// SIMATIC S7-200 project (STEP 7-Micro/WIN), CPU 226 REL 02.01

SYMBOL_TABLE USR1
出水温度VF           I0.0
回水温度VF           I0.1
燃烧信号             I0.2
尾烟温度VF           I0.3
超温报警             I0.4
超高压力             I0.5
低限压力             I0.6
循环泵信号            I0.7
风机反馈             I1.0
低水位              I1.1
停炉消音             I1.2
熄火               I1.3
启动复位             I1.4
循环水泵             Q0.0
蜂鸣器              Q0.1
风机               Q0.2
减低负荷             Q0.4
加大负荷             Q0.5
锅炉运行控制           Q0.7
故障               Q1.0
第一段温度            M0.0
第二段温度            M0.1
第三段温度            M0.2
第四段温度            M0.3
第五段温度            M0.4
显示手动键            M1.4
后扫显示             M1.5
强制小火显示           M1.6
复位显示             M1.7
点火成功             M2.0
可以燃烧             M2.1
喷油标志             M2.4
进入消音             M2.6
停火消音             M2.7
手动负荷             M4.0
手动关小             M4.1
手动开大             M4.2
分段控制             M4.5
工作时间             M4.6
等待工作             M5.0
启动标志             M5.1
锅炉启动             M5.2
停火标志             M5.7
负荷减小             M6.0
负荷加大             M6.1
负荷在减小            M6.2
负荷在加大            M6.3
消音标志             M7.3
屏启动按钮            M8.0
屏停炉按钮            M8.1
屏消音按钮            M8.2
屏复位按钮            M8.3
消音脉冲             M8.5
启动脉冲             M8.6
复位脉冲             M8.7
PLC是运行           M9.0
记录清零             M9.3
停火故障             M9.6
严重故障             M9.7
报极低水位            M10.7
锅炉压力失常           M10.6
传感器故障            M10.5
报限位故障            M10.4
报超高温度            M10.3
风门关故障            M10.2
风门中继坏            M10.1
燃气压力低            M10.0
超高烟温             M11.7
点火失败             M11.6
风压不足故障           M11.5
关阀故障             M11.4
故障熄火             M11.3
故障见火             M11.2
风门开故障            M11.1
风门小故障            M11.0
要求大火             M12.2
记录小火             M12.3
动画小火             M12.4
记录大火             M12.5
动画大火             M12.6
温度启停炉            M13.1
出口传感器故障          M13.2
烟温高              M13.3
大小火控制            M13.5
设置时间             M14.0
不检传感             M14.4
管理密码对            M15.1
MODBUS1          M18.0
MODBUS2          M18.1
屏动画风机            M20.0
屏动画水泵            M20.1
强制小火             M31.1
手动开风机            M31.2
水泵自动             M31.3
水泵手动             M31.4
水泵停              M31.5
PLC运行            SM0.0
运行脉冲             SM0.1
分振荡器             SM0.4
PLC在运行           SM0.7
中断1              SMB34
中断2              SMB35
HC0控制字           SMB37
HC0当前值           SMD38
HC3控制字           SMB137
HC3当前值           SMD138
HC4控制字           SMB147
HC4当前值           SMD148
不见光极限            T34
确认点火             T37
确认停火             T38
确认小火             T42
报警延时             T49
是极低水位            T51
是超高温度            T52
是锅炉超压            T53
是欠压              T54
是传感器故障           T55
是烟温高             T56
减负荷              T101
加负荷              T102
开机3秒             T103
后吹扫控制            T112
程控小火完成           T117
报荡显示1            T130
振荡显示2            T131
开机2秒             T142
记录工时分            C15
水泵工时分            C16
风机工时分            C17
燃烧工时分            C18
时间（年）16          VB10
时间（月）16          VB11
时间（日）16          VB12
时间（时）16          VB13
时间（分）16          VB14
时间（秒）16          VB15
实际状态编码           VW18
密码确认1            VW20
密码确认2            VW22
密码确认3            VW24
密码确认4            VW26
时间分段数            VW38
后吹扫时间            VW40
强制小火时间           VW46
给定出口温度           VD50
给定出口温度W          VW52
给定尾烟温            VW54
禁改测试页号           VW58
开机密码             VW62
管理密码             VW64
输管理密码            VW66
输开机密码            VW68
MODBUS11         VB70
MODBUS21         VB71
实际工作段            VB72
屏火焰指针            VW82
故障编码             VW86
高8               VB88
低8               VB89
故障码反             VW88
出口截距             VW90
回水截距             VW92
尾烟截距             VW94
启炉温              VW96
停火温              VW98
出口斜率             VD100
回水斜率             VD104
尾烟斜率             VD108
设定停火温            VW120
设定启动温            VW122
点火次数             VW140
工时               VW142
停炉故障次            VW144
低水位故障次           VW146
熄火次数             VW148
高温停炉次            VW150
水泵工时             VW160
风机工时             VW162
燃烧工时             VW164
定时控制             VW200
积分加强             VD202
微分加强             VD212
EI               VD222
EI1              VD232
EI2              VD242
AEI              VD252
AEI1             VD262
AAEI             VD272
查EI              VD282
比例加强             VD292
负荷调节总量           VD302
比例计算             VD312
P                VD322
积分计算             VD332
I                VD342
微分计算             VD352
D                VD362
PID计算            VD372
PID              VD382
PID累加            VD392
可控PID            VD402
余下PID            VD412
正PID控制时间         VD422
加PID             VW424
剩余PID            VD432
负PID控制时间         VD442
减PID             VW444
普通出口设定温          VD900
第一时间段设定温度1       VD904
第二时间段设定温度2       VD908
第三时间段设定温度3       VD912
第四时间段设定温度4       VD916
第五时间段设定温度5       VD920
采样记数器            VW1000
实际出口温            VD1020
实际出口温W           VW1022
出口温采样值           VD1024
出口采样             VW1026
出水计算1            VD1032
出水计算1高8位         VW1032
出水计算1低8位         VW1034
出水计算2            VD1036
实际回水温            VD1040
实际回水温W           VW1042
回水温采样值           VD1044
回水采样             VW1046
回水计算1            VD1052
回水计算1高8位         VW1052
回水计算1低8位         VW1054
回水计算2            VD1056
实际尾烟温            VD1060
实际尾烟温W           VW1062
尾烟温采样值           VD1064
尾烟采样             VW1066
尾烟计算1            VD1072
尾烟计算1高8位         VW1072
尾烟计算1低8位         VW1074
尾烟计算2            VD1076
时间1开时            VW2370
时间1开分            VW2376
时间1关时            VW2390
时间1关分            VW2396
时间2开时            VW2410
时间2开分            VW2416
时间2关时            VW2430
时间2关分            VW2436
时间3开时            VW2450
时间3开分            VW2456
时间3关时            VW2470
时间3关分            VW2476
时间4开时            VW2490
时间4开分            VW2496
时间4关时            VW2510
时间4关分            VW2516
时间5开时            VW2530
时间5开分            VW2536
时间5关时            VW2550
时间5关分            VW2556
实际时间             VW2600
实际时              VW2602
实际分              VW2604
实际时转分            VW2606
开1时间             VW2610
开1时转分            VW2612
关1时间             VW2616
关1时转分            VW2618
开2时间             VW2620
开2时转分            VW2622
关2时间             VW2626
关2时转分            VW2628
开3时间             VW2630
开3时转分            VW2632
关3时间             VW2636
关3时转分            VW2638
开4时间             VW2640
开4时转分            VW2642
关4时间             VW2646
关4时转分            VW2648
开5时间             VW2650
开5时转分            VW2652
关5时间             VW2656
关5时转分            VW2658
传送首址             VB3000
传工作状态            VW3000
传极低水位            VW3002
传锅炉压力失常          VW3004
传出口传感故障          VW3006
传燃烧器限位故障         VW3008
传超高温度            VW3010
传风门关闭故障          VW3012
传风门中继故障          VW3014
传燃气压力低           VW3016
传超高烟温            VW3018
传风压不足            VW3020
传关阀故障            VW3022
传熄火故障            VW3024
传故障见火            VW3026
传风门开故障           VW3028
传风门小故障           VW3030
传后扫时间            VW3032
传强制小火时间          VW3034
传点火次数            VW3036
传工时              VW3038
传故障停炉次数          VW3040
传给定温度            VW3042
传给定烟温            VW3044
传实际烟温            VW3046
传实际出口温           VW3048
传实际回水温           VW3050
END_SYMBOL_TABLE

SYMBOL_TABLE USS Protocol
USS_LOW_V        VD1000   // (DWORD) Enter the starting address for USS Protocol symbols here.
USS_HIGH_V       VD1004
USS_TIME_OUT     VW1008
USS_I_LINE       VW1010
USS_DAT_PTR0     VD1012
USS_ACT_DRV0     VD1016
USS_CUR_DRV0     VD1020
USS_P0           V1024.0
USS_REQ_SNT0     V1024.1
USS_RETRY_P0     VB1025
USS_ERR_CODE     VB1026
USS_CS_D0        VD1027
USS_CS_W0        VW1027
USS_CS_W2        VW1029
USS_CS_B0        VB1027
USS_CS_B1        VB1028
USS_POLL_BUF     VB1031
USS_XMT_0        VB1046
USS_XMT_ADR0     VB1049
USS_X_STWD       VD1056
USS_X_BCC        VB1060
USS_X_DW1        VD1047
USS_X_DW5        VD1051
USS_X_DW9        VD1055
USS_X_DB13       VB1059
USS_RCV_BUF0     VB1061
USS_R_STX        VB1062
USS_R_LGE        VB1063
USS_R_ADR        VB1064
USS_R_STWD       VD1071
USS_R_DW1        VD1062
USS_R_DW5        VD1066
USS_R_DW9        VD1070
USS_R_W13        VW1074
USS_STAT_TAB     VB1076
USS_ADR_P0       VB1396
END_SYMBOL_TABLE

ORGANIZATION_BLOCK MAIN:OB1
TITLE= 
// PROGRAM COMMENTS
// Press F1 for help and example program
//  
BEGIN
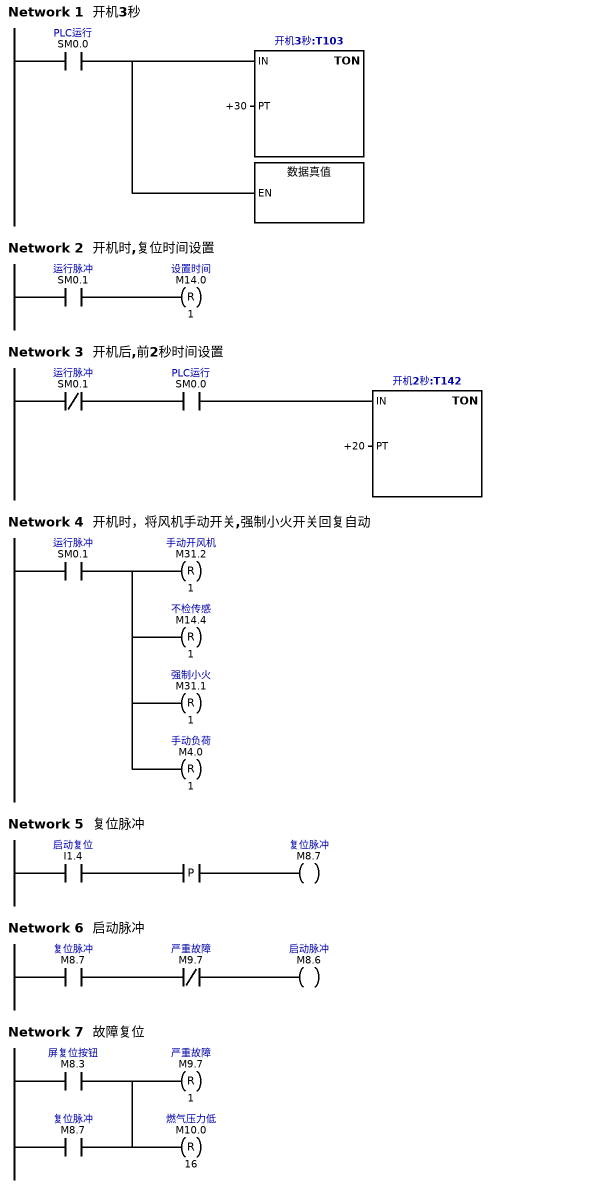
Network 1 // 开机3秒
// 
// 
LD     PLC运行:SM0.0
TON    开机3秒:T103, +30
CALL   数据真值:SBR0
Network 2 // 开机时,复位时间设置
LD     运行脉冲:SM0.1
R      设置时间:M14.0, 1
Network 3 // 开机后,前2秒时间设置
// 
// 
LDN    运行脉冲:SM0.1
A      PLC运行:SM0.0
TON    开机2秒:T142, +20
Network 4 // 开机时，将风机手动开关,强制小火开关回复自动
// 
// 
LD     运行脉冲:SM0.1
R      手动开风机:M31.2, 1
R      不检传感:M14.4, 1
R      强制小火:M31.1, 1
R      手动负荷:M4.0, 1
Network 5 // 复位脉冲
LD     启动复位:I1.4
EU
=      复位脉冲:M8.7
Network 6 // 启动脉冲
LD     复位脉冲:M8.7
AN     严重故障:M9.7
=      启动脉冲:M8.6
Network 7 // 故障复位
// 
// 
LD     屏复位按钮:M8.3
O      复位脉冲:M8.7
R      严重故障:M9.7, 1
R      燃气压力低:M10.0, 16
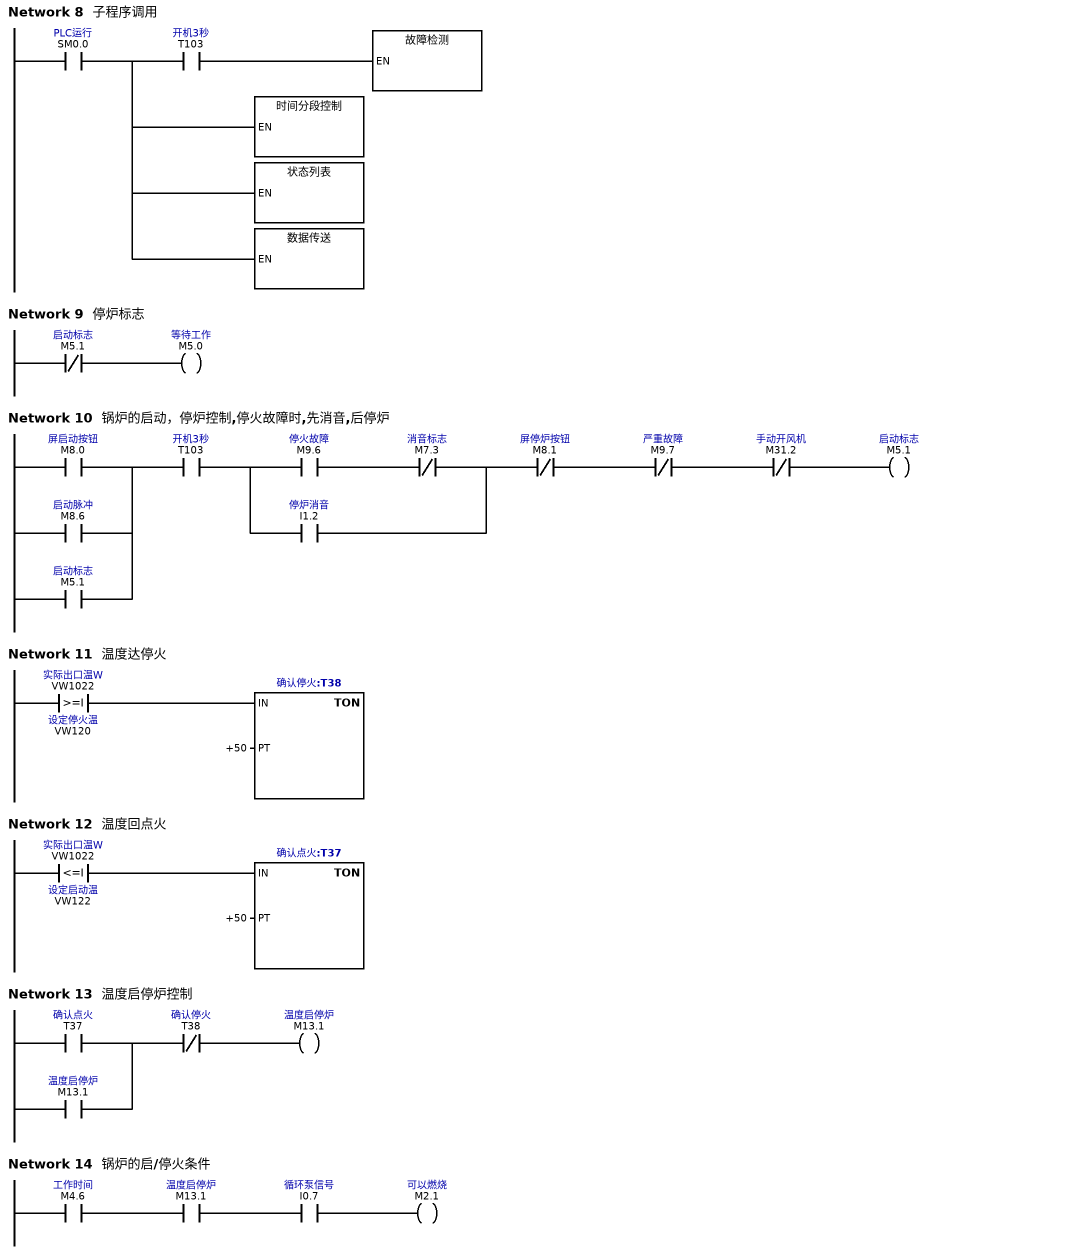
Network 8 // 子程序调用
// 
//  
LD     PLC运行:SM0.0
LPS
A      开机3秒:T103
CALL   故障检测:SBR4
LRD
CALL   时间分段控制:SBR6
LRD
CALL   状态列表:SBR7
LPP
CALL   数据传送:SBR8
Network 9 // 停炉标志
// 
// 
LDN    启动标志:M5.1
=      等待工作:M5.0
Network 10 // 锅炉的启动，停炉控制,停火故障时,先消音,后停炉
// 
// 
LD     屏启动按钮:M8.0
O      启动脉冲:M8.6
O      启动标志:M5.1
A      开机3秒:T103
LD     停火故障:M9.6
AN     消音标志:M7.3
O      停炉消音:I1.2
ALD
AN     屏停炉按钮:M8.1
AN     严重故障:M9.7
AN     手动开风机:M31.2
=      启动标志:M5.1
Network 11 // 温度达停火
// 
// 
LDW>=  实际出口温W:VW1022, 设定停火温:VW120
TON    确认停火:T38, +50
Network 12 // 温度回点火
// 
// 
LDW<=  实际出口温W:VW1022, 设定启动温:VW122
TON    确认点火:T37, +50
Network 13 // 温度启停炉控制
// 
// 
LD     确认点火:T37
O      温度启停炉:M13.1
AN     确认停火:T38
=      温度启停炉:M13.1
Network 14 // 锅炉的启/停火条件
// 
// 
LD     工作时间:M4.6
A      温度启停炉:M13.1
A      循环泵信号:I0.7
=      可以燃烧:M2.1
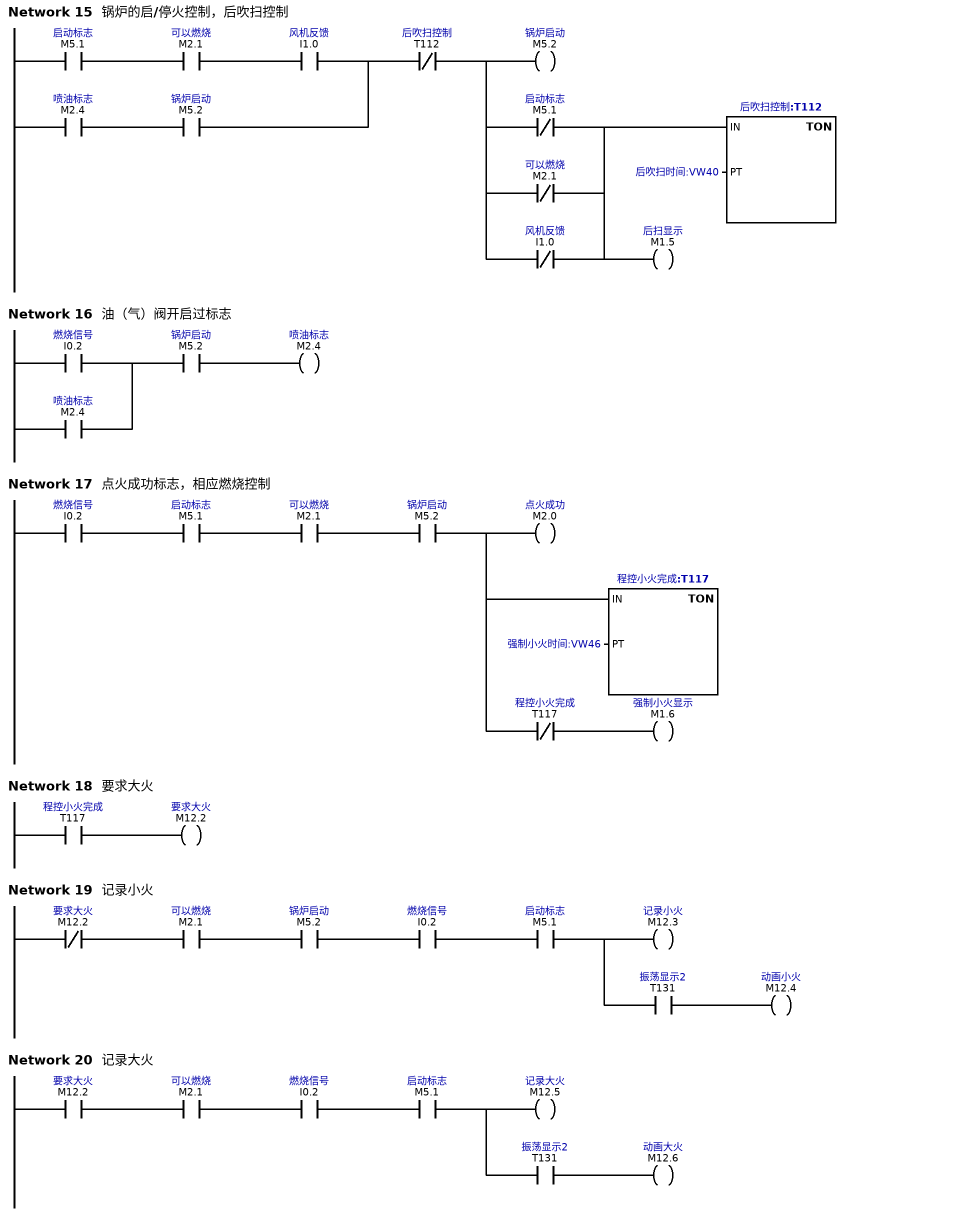
Network 15 // 锅炉的启/停火控制，后吹扫控制
// 
// 
LD     启动标志:M5.1
A      可以燃烧:M2.1
A      风机反馈:I1.0
LD     喷油标志:M2.4
A      锅炉启动:M5.2
OLD
AN     后吹扫控制:T112
=      锅炉启动:M5.2
LDN    启动标志:M5.1
ON     可以燃烧:M2.1
ON     风机反馈:I1.0
ALD
TON    后吹扫控制:T112, 后吹扫时间:VW40
=      后扫显示:M1.5
Network 16 // 油（气）阀开启过标志
// 
// 
LD     燃烧信号:I0.2
O      喷油标志:M2.4
A      锅炉启动:M5.2
=      喷油标志:M2.4
Network 17 // 点火成功标志，相应燃烧控制
// 
// 
LD     燃烧信号:I0.2
A      启动标志:M5.1
A      可以燃烧:M2.1
A      锅炉启动:M5.2
=      点火成功:M2.0
TON    程控小火完成:T117, 强制小火时间:VW46
AN     程控小火完成:T117
=      强制小火显示:M1.6
Network 18 // 要求大火
LD     程控小火完成:T117
=      要求大火:M12.2
Network 19 // 记录小火
LDN    要求大火:M12.2
A      可以燃烧:M2.1
A      锅炉启动:M5.2
A      燃烧信号:I0.2
A      启动标志:M5.1
=      记录小火:M12.3
A      振荡显示2:T131
=      动画小火:M12.4
Network 20 // 记录大火
LD     要求大火:M12.2
A      可以燃烧:M2.1
A      燃烧信号:I0.2
A      启动标志:M5.1
=      记录大火:M12.5
A      振荡显示2:T131
=      动画大火:M12.6
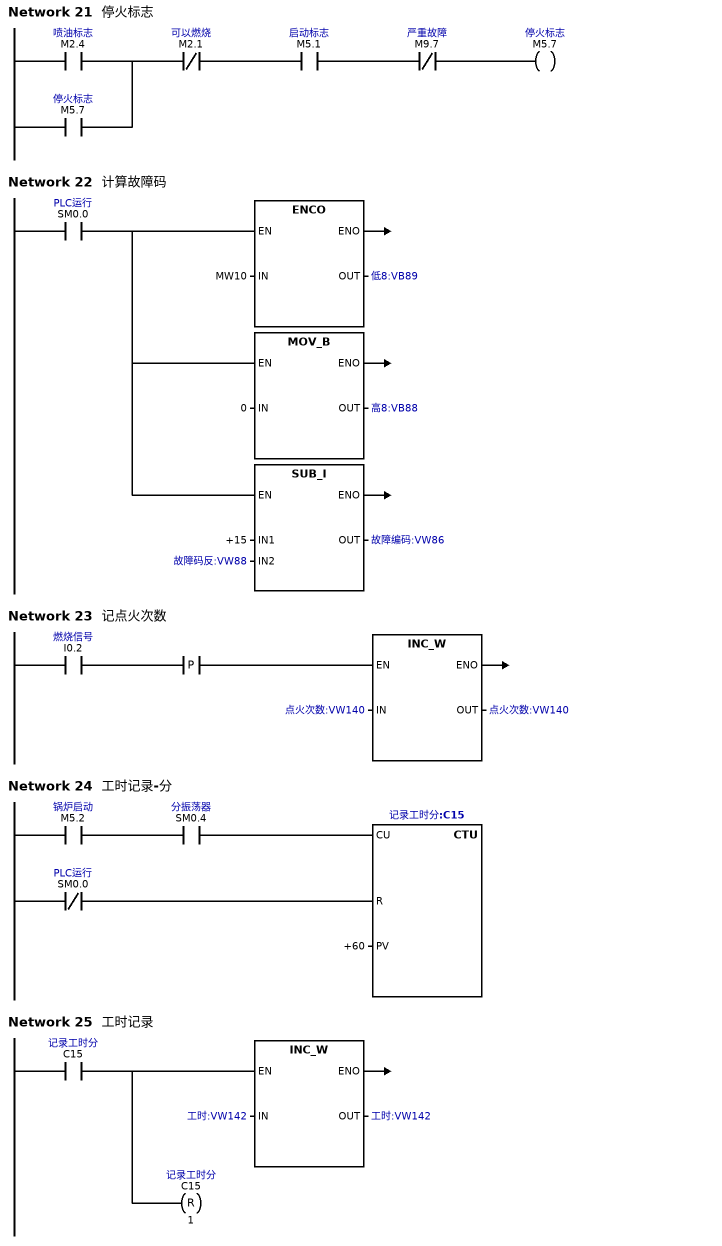
Network 21 // 停火标志
// 
// 
LD     喷油标志:M2.4
O      停火标志:M5.7
AN     可以燃烧:M2.1
A      启动标志:M5.1
AN     严重故障:M9.7
=      停火标志:M5.7
Network 22 // 计算故障码
// 
// 
LD     PLC运行:SM0.0
ENCO   MW10, 低8:VB89
MOVB   0, 高8:VB88
MOVW   +15, 故障编码:VW86
-I     故障码反:VW88, 故障编码:VW86
Network 23 // 记点火次数
// 
// 
LD     燃烧信号:I0.2
EU
INCW   点火次数:VW140
Network 24 // 工时记录-分
// 
// 
LD     锅炉启动:M5.2
A      分振荡器:SM0.4
LDN    PLC运行:SM0.0
CTU    记录工时分:C15, +60
Network 25 // 工时记录
// 
// 
LD     记录工时分:C15
INCW   工时:VW142
R      记录工时分:C15, 1
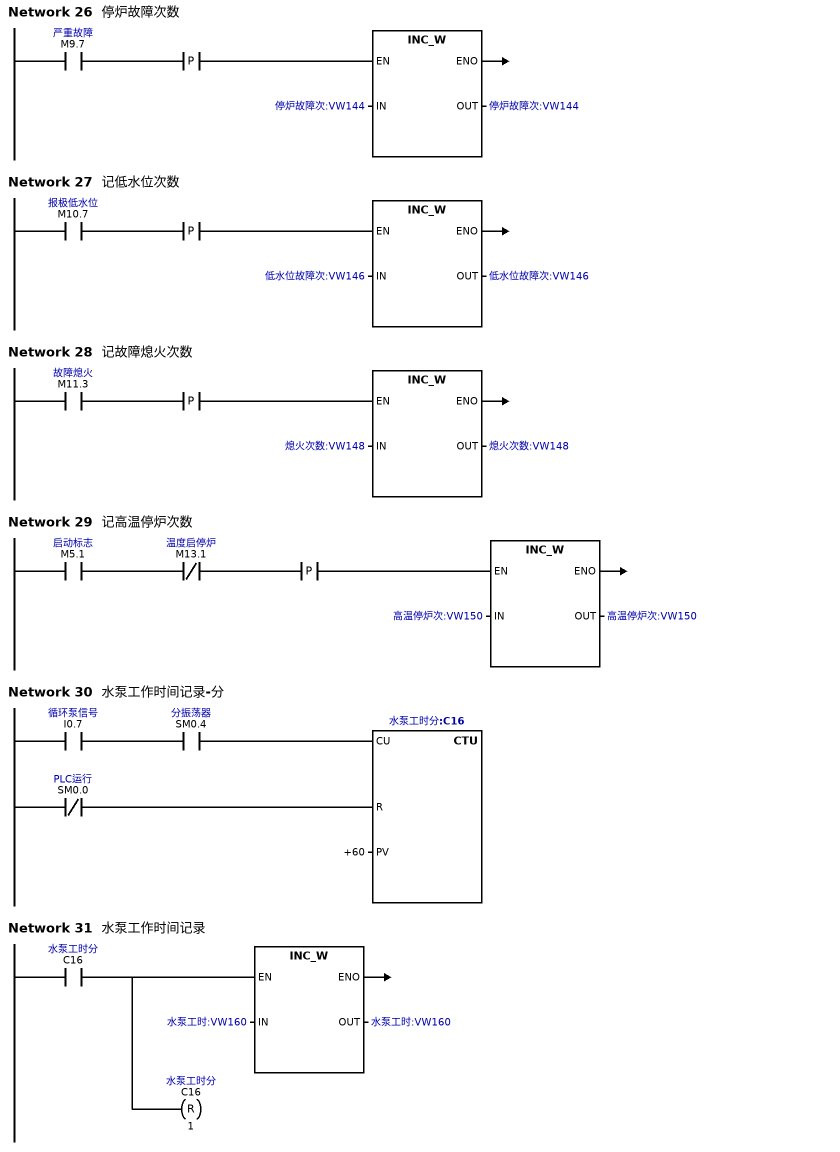
Network 26 // 停炉故障次数
// 
// 
LD     严重故障:M9.7
EU
INCW   停炉故障次:VW144
Network 27 // 记低水位次数
// 
// 
LD     报极低水位:M10.7
EU
INCW   低水位故障次:VW146
Network 28 // 记故障熄火次数
// 
// 
LD     故障熄火:M11.3
EU
INCW   熄火次数:VW148
Network 29 // 记高温停炉次数
// 
// 
LD     启动标志:M5.1
AN     温度启停炉:M13.1
EU
INCW   高温停炉次:VW150
Network 30 // 水泵工作时间记录-分
// 
// 
LD     循环泵信号:I0.7
A      分振荡器:SM0.4
LDN    PLC运行:SM0.0
CTU    水泵工时分:C16, +60
Network 31 // 水泵工作时间记录
// 
// 
LD     水泵工时分:C16
INCW   水泵工时:VW160
R      水泵工时分:C16, 1
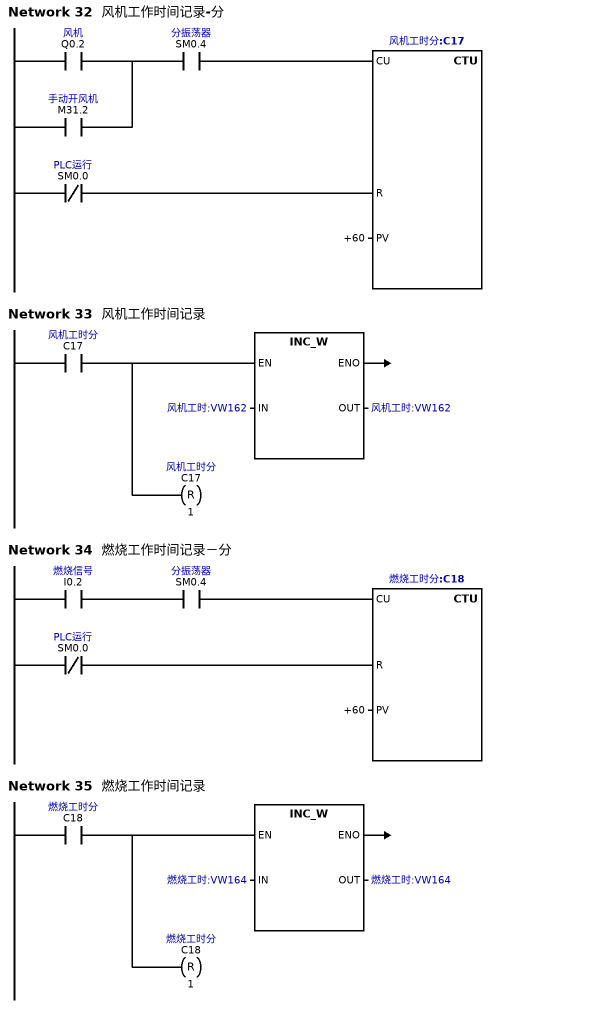
Network 32 // 风机工作时间记录-分
// 
// 
LD     风机:Q0.2
O      手动开风机:M31.2
A      分振荡器:SM0.4
LDN    PLC运行:SM0.0
CTU    风机工时分:C17, +60
Network 33 // 风机工作时间记录
// 
// 
LD     风机工时分:C17
INCW   风机工时:VW162
R      风机工时分:C17, 1
Network 34 // 燃烧工作时间记录－分
// 
// 
LD     燃烧信号:I0.2
A      分振荡器:SM0.4
LDN    PLC运行:SM0.0
CTU    燃烧工时分:C18, +60
Network 35 // 燃烧工作时间记录
// 
// 
LD     燃烧工时分:C18
INCW   燃烧工时:VW164
R      燃烧工时分:C18, 1
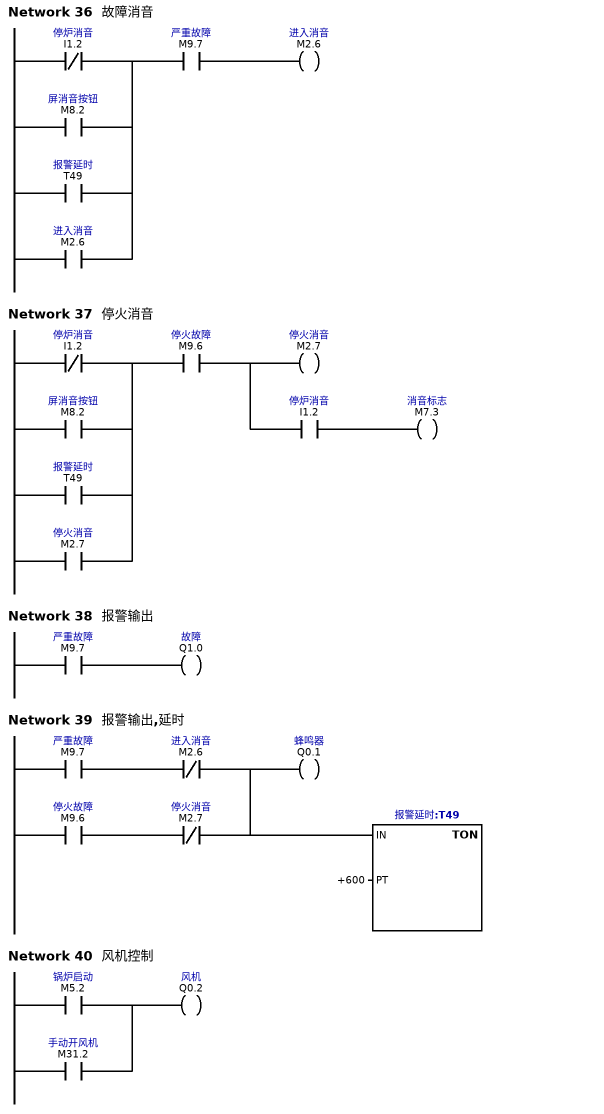
Network 36 // 故障消音
LDN    停炉消音:I1.2
O      屏消音按钮:M8.2
O      报警延时:T49
O      进入消音:M2.6
A      严重故障:M9.7
=      进入消音:M2.6
Network 37 // 停火消音
LDN    停炉消音:I1.2
O      屏消音按钮:M8.2
O      报警延时:T49
O      停火消音:M2.7
A      停火故障:M9.6
=      停火消音:M2.7
A      停炉消音:I1.2
=      消音标志:M7.3
Network 38 // 报警输出
// 
// 
LD     严重故障:M9.7
=      故障:Q1.0
Network 39 // 报警输出,延时
// 
// 
LD     严重故障:M9.7
AN     进入消音:M2.6
LD     停火故障:M9.6
AN     停火消音:M2.7
OLD
=      蜂鸣器:Q0.1
TON    报警延时:T49, +600
Network 40 // 风机控制
// 
// 
LD     锅炉启动:M5.2
O      手动开风机:M31.2
=      风机:Q0.2
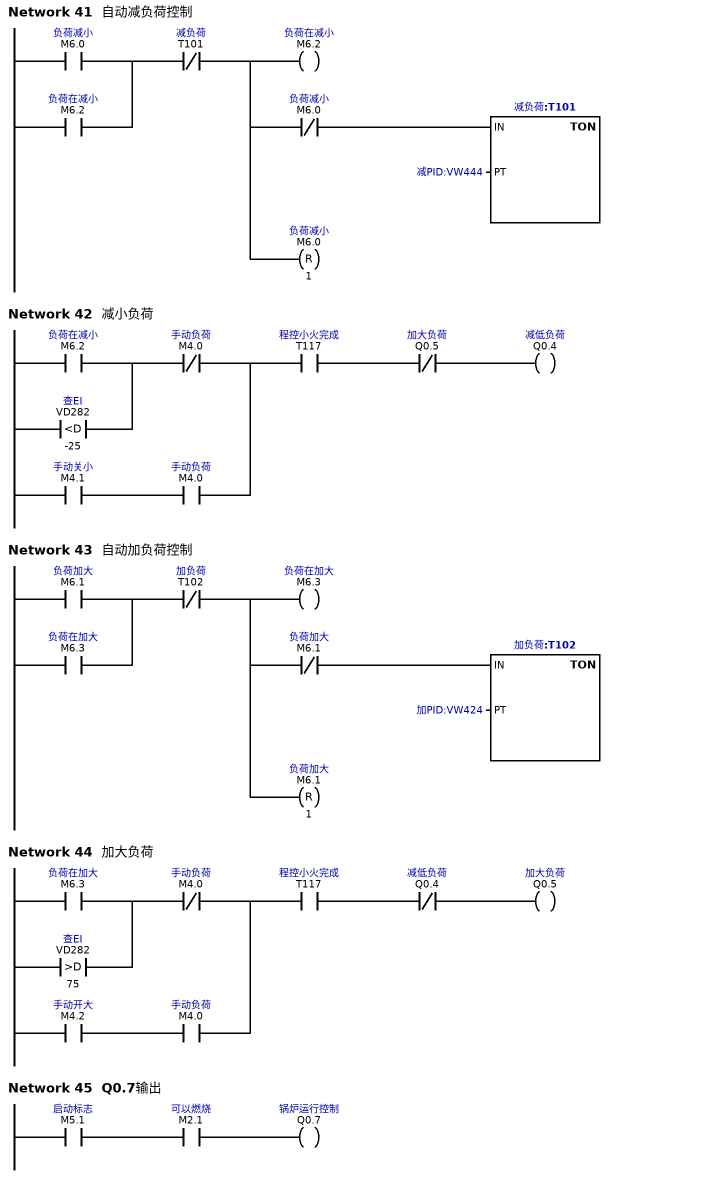
Network 41 // 自动减负荷控制
LD     负荷减小:M6.0
O      负荷在减小:M6.2
AN     减负荷:T101
LPS
=      负荷在减小:M6.2
AN     负荷减小:M6.0
TON    减负荷:T101, 减PID:VW444
LPP
R      负荷减小:M6.0, 1
Network 42 // 减小负荷
LD     负荷在减小:M6.2
OD<    查EI:VD282, -25
AN     手动负荷:M4.0
LD     手动关小:M4.1
A      手动负荷:M4.0
OLD
A      程控小火完成:T117
AN     加大负荷:Q0.5
=      减低负荷:Q0.4
Network 43 // 自动加负荷控制
LD     负荷加大:M6.1
O      负荷在加大:M6.3
AN     加负荷:T102
LPS
=      负荷在加大:M6.3
AN     负荷加大:M6.1
TON    加负荷:T102, 加PID:VW424
LPP
R      负荷加大:M6.1, 1
Network 44 // 加大负荷
// 
// 
LD     负荷在加大:M6.3
OD>    查EI:VD282, 75
AN     手动负荷:M4.0
LD     手动开大:M4.2
A      手动负荷:M4.0
OLD
A      程控小火完成:T117
AN     减低负荷:Q0.4
=      加大负荷:Q0.5
Network 45 // Q0.7输出
// 
// 
LD     启动标志:M5.1
A      可以燃烧:M2.1
=      锅炉运行控制:Q0.7
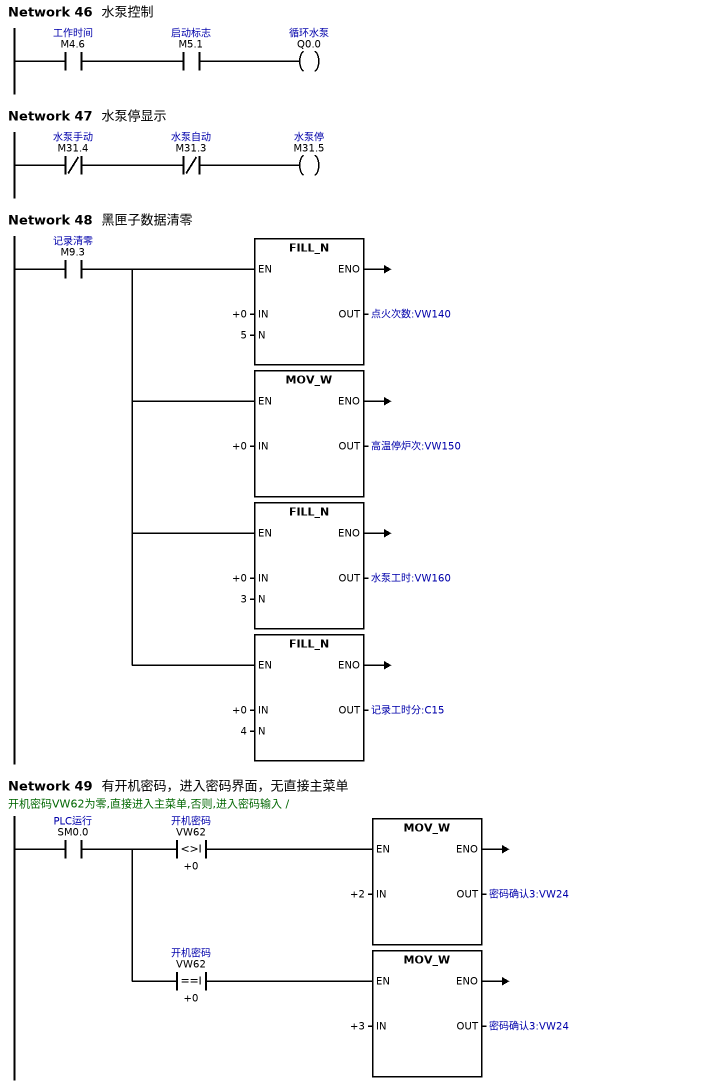
Network 46 // 水泵控制
// 
// 
LD     工作时间:M4.6
A      启动标志:M5.1
=      循环水泵:Q0.0
Network 47 // 水泵停显示
// 
// 
LDN    水泵手动:M31.4
AN     水泵自动:M31.3
=      水泵停:M31.5
Network 48 // 黑匣子数据清零
// 
// 
LD     记录清零:M9.3
FILL   +0, 点火次数:VW140, 5
MOVW   +0, 高温停炉次:VW150
FILL   +0, 水泵工时:VW160, 3
FILL   +0, 记录工时分:C15, 4
Network 49 // 有开机密码，进入密码界面，无直接主菜单
// 开机密码VW62为零,直接进入主菜单,否则,进入密码输入
// 
LD     PLC运行:SM0.0
LPS
AW<>   开机密码:VW62, +0
MOVW   +2, 密码确认3:VW24
LPP
AW=    开机密码:VW62, +0
MOVW   +3, 密码确认3:VW24
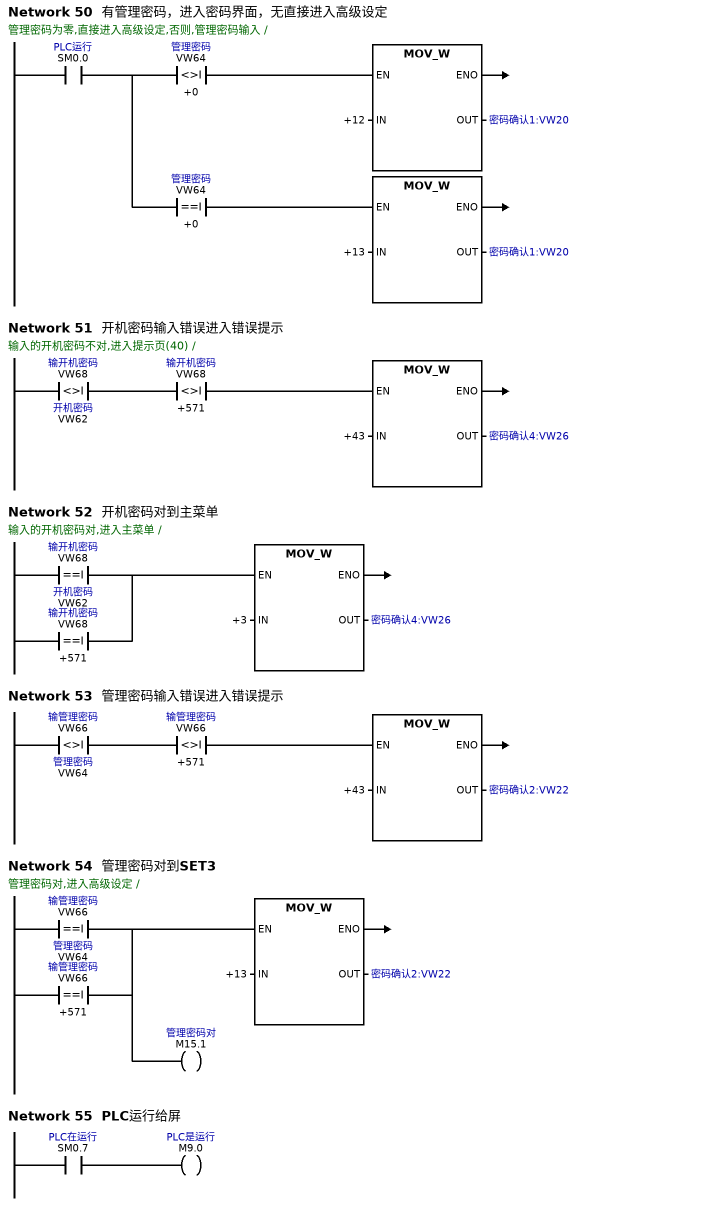
Network 50 // 有管理密码，进入密码界面，无直接进入高级设定
// 管理密码为零,直接进入高级设定,否则,管理密码输入
// 
LD     PLC运行:SM0.0
LPS
AW<>   管理密码:VW64, +0
MOVW   +12, 密码确认1:VW20
LPP
AW=    管理密码:VW64, +0
MOVW   +13, 密码确认1:VW20
Network 51 // 开机密码输入错误进入错误提示
// 输入的开机密码不对,进入提示页(40)
// 
LDW<>  输开机密码:VW68, 开机密码:VW62
AW<>   输开机密码:VW68, +571
MOVW   +43, 密码确认4:VW26
Network 52 // 开机密码对到主菜单
// 输入的开机密码对,进入主菜单
// 
LDW=   输开机密码:VW68, 开机密码:VW62
OW=    输开机密码:VW68, +571
MOVW   +3, 密码确认4:VW26
Network 53 // 管理密码输入错误进入错误提示
// 
// 
LDW<>  输管理密码:VW66, 管理密码:VW64
AW<>   输管理密码:VW66, +571
MOVW   +43, 密码确认2:VW22
Network 54 // 管理密码对到SET3
// 管理密码对,进入高级设定
// 
LDW=   输管理密码:VW66, 管理密码:VW64
OW=    输管理密码:VW66, +571
MOVW   +13, 密码确认2:VW22
=      管理密码对:M15.1
Network 55 // PLC运行给屏
// 
// 
LD     PLC在运行:SM0.7
=      PLC是运行:M9.0
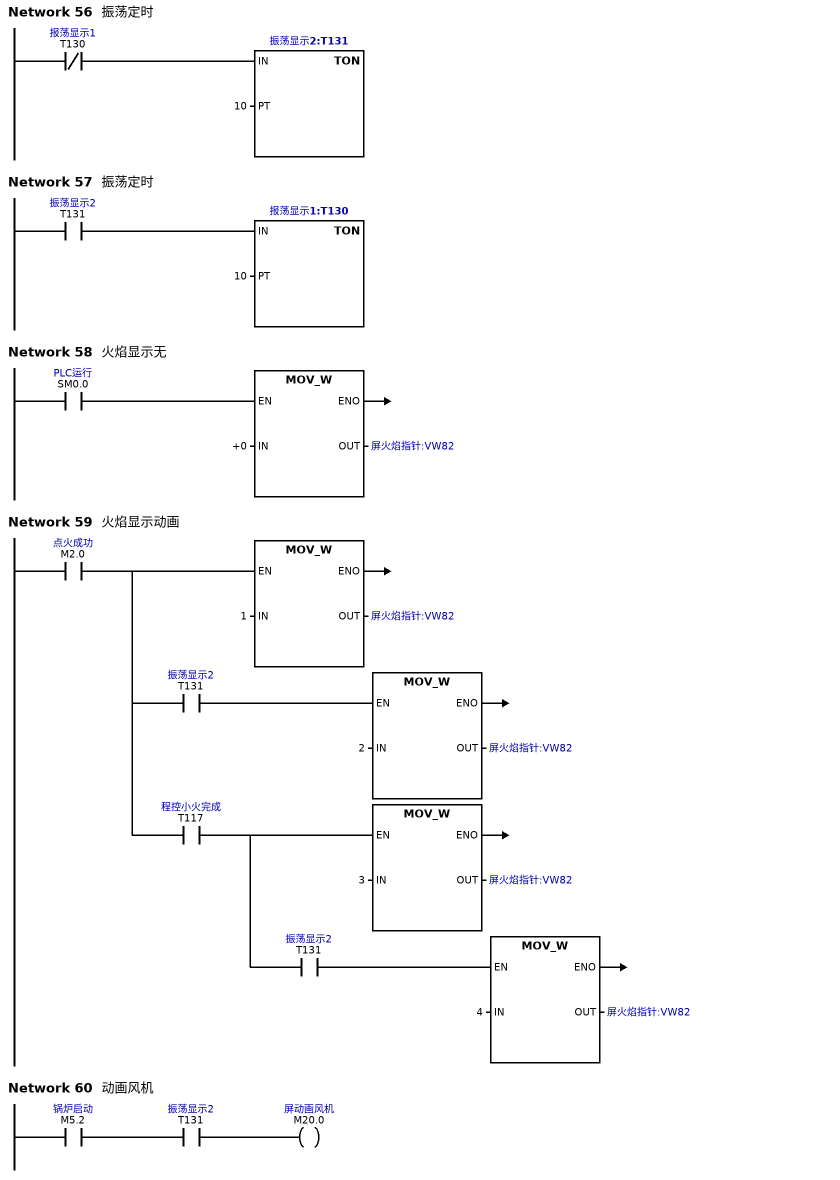
Network 56 // 振荡定时
// 
// 
LDN    报荡显示1:T130
TON    振荡显示2:T131, 10
Network 57 // 振荡定时
// 
// 
LD     振荡显示2:T131
TON    报荡显示1:T130, 10
Network 58 // 火焰显示无
// 
// 
LD     PLC运行:SM0.0
MOVW   +0, 屏火焰指针:VW82
Network 59 // 火焰显示动画
// 
// 
LD     点火成功:M2.0
LPS
MOVW   1, 屏火焰指针:VW82
A      振荡显示2:T131
MOVW   2, 屏火焰指针:VW82
LPP
A      程控小火完成:T117
MOVW   3, 屏火焰指针:VW82
A      振荡显示2:T131
MOVW   4, 屏火焰指针:VW82
Network 60 // 动画风机
// 
// 
LD     锅炉启动:M5.2
A      振荡显示2:T131
=      屏动画风机:M20.0
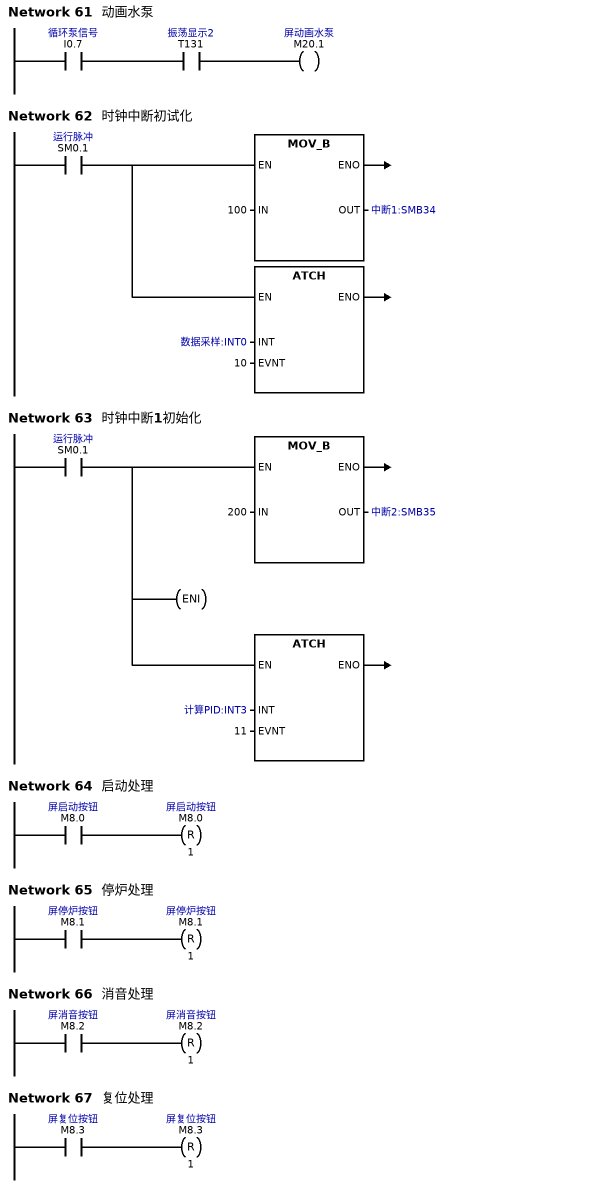
Network 61 // 动画水泵
// 
// 
LD     循环泵信号:I0.7
A      振荡显示2:T131
=      屏动画水泵:M20.1
Network 62 // 时钟中断初试化
// 
// 
LD     运行脉冲:SM0.1
MOVB   100, 中断1:SMB34
ATCH   数据采样:INT0, 10
Network 63 // 时钟中断1初始化
LD     运行脉冲:SM0.1
MOVB   200, 中断2:SMB35
ENI
ATCH   计算PID:INT3, 11
Network 64 // 启动处理
LD     屏启动按钮:M8.0
R      屏启动按钮:M8.0, 1
Network 65 // 停炉处理
LD     屏停炉按钮:M8.1
R      屏停炉按钮:M8.1, 1
Network 66 // 消音处理
LD     屏消音按钮:M8.2
R      屏消音按钮:M8.2, 1
Network 67 // 复位处理
LD     屏复位按钮:M8.3
R      屏复位按钮:M8.3, 1
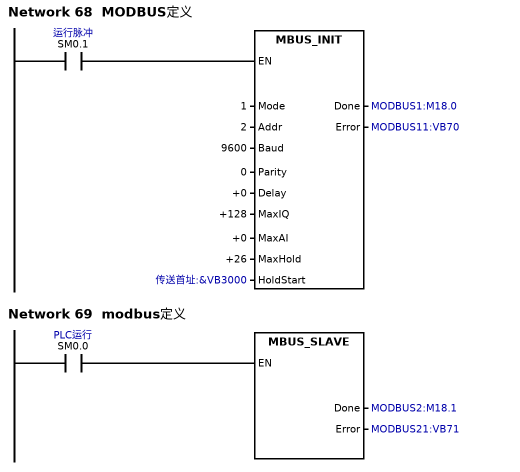
Network 68 // MODBUS定义
LD     运行脉冲:SM0.1
CALL   MBUS_INIT:SBR1, 1, 2, 9600, 0, +0, +128, +0, +26, &传送首址:VB3000, MODBUS1:M18.0, MODBUS11:VB70
Network 69 // modbus定义
LD     PLC运行:SM0.0
CALL   MBUS_SLAVE:SBR2, MODBUS2:M18.1, MODBUS21:VB71
END_ORGANIZATION_BLOCK

SUBROUTINE_BLOCK 数据真值:SBR0
TITLE= 
// SUBROUTINE COMMENTS
// Press F1 for help and example program
//  
BEGIN
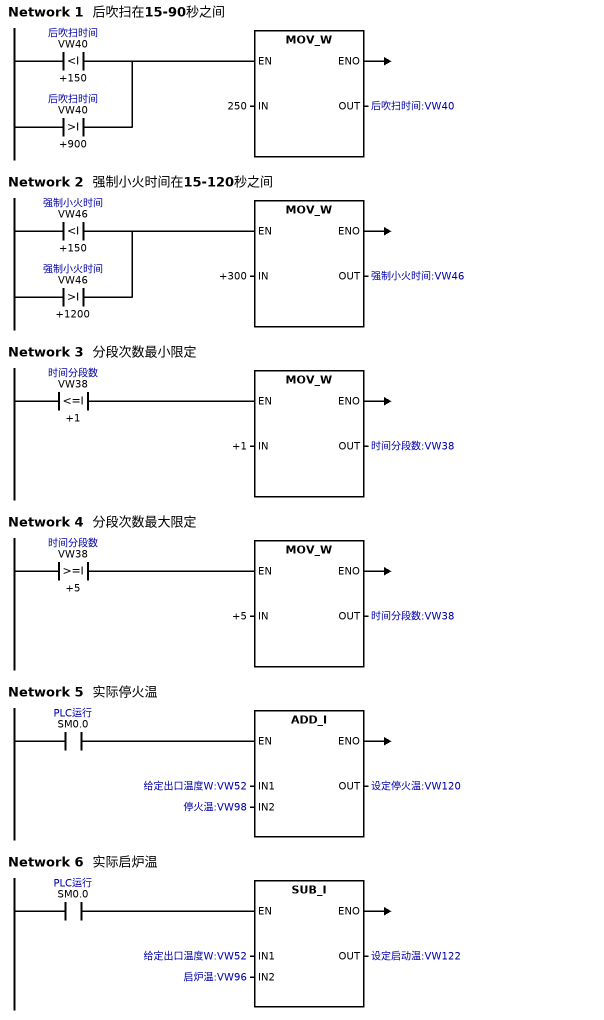
Network 1 // 后吹扫在15-90秒之间
// 
// 
LDW<   后吹扫时间:VW40, +150
OW>    后吹扫时间:VW40, +900
MOVW   250, 后吹扫时间:VW40
Network 2 // 强制小火时间在15-120秒之间
// 
// 
LDW<   强制小火时间:VW46, +150
OW>    强制小火时间:VW46, +1200
MOVW   +300, 强制小火时间:VW46
Network 3 // 分段次数最小限定
// 
// 
LDW<=  时间分段数:VW38, +1
MOVW   +1, 时间分段数:VW38
Network 4 // 分段次数最大限定
// 
// 
LDW>=  时间分段数:VW38, +5
MOVW   +5, 时间分段数:VW38
Network 5 // 实际停火温
// 
// 
LD     PLC运行:SM0.0
MOVW   给定出口温度W:VW52, 设定停火温:VW120
+I     停火温:VW98, 设定停火温:VW120
Network 6 // 实际启炉温
// 
// 
LD     PLC运行:SM0.0
MOVW   给定出口温度W:VW52, 设定启动温:VW122
-I     启炉温:VW96, 设定启动温:VW122
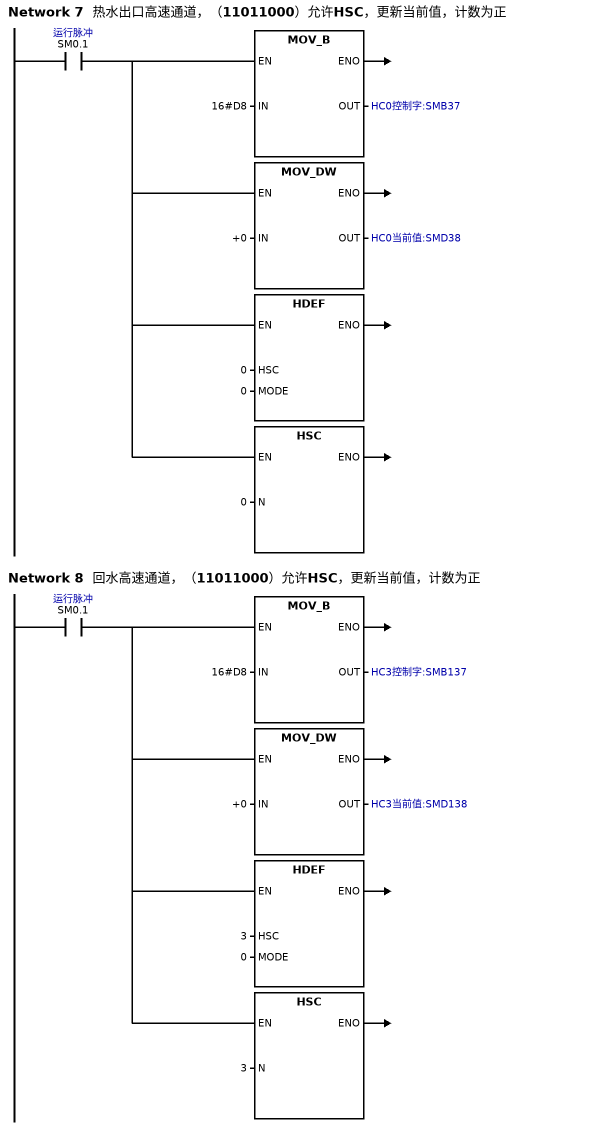
Network 7 // 热水出口高速通道，（11011000）允许HSC，更新当前值，计数为正
// 
// 
LD     运行脉冲:SM0.1
MOVB   16#D8, HC0控制字:SMB37
MOVD   +0, HC0当前值:SMD38
HDEF   0, 0
HSC    0
Network 8 // 回水高速通道，（11011000）允许HSC，更新当前值，计数为正
// 
// 
LD     运行脉冲:SM0.1
MOVB   16#D8, HC3控制字:SMB137
MOVD   +0, HC3当前值:SMD138
HDEF   3, 0
HSC    3
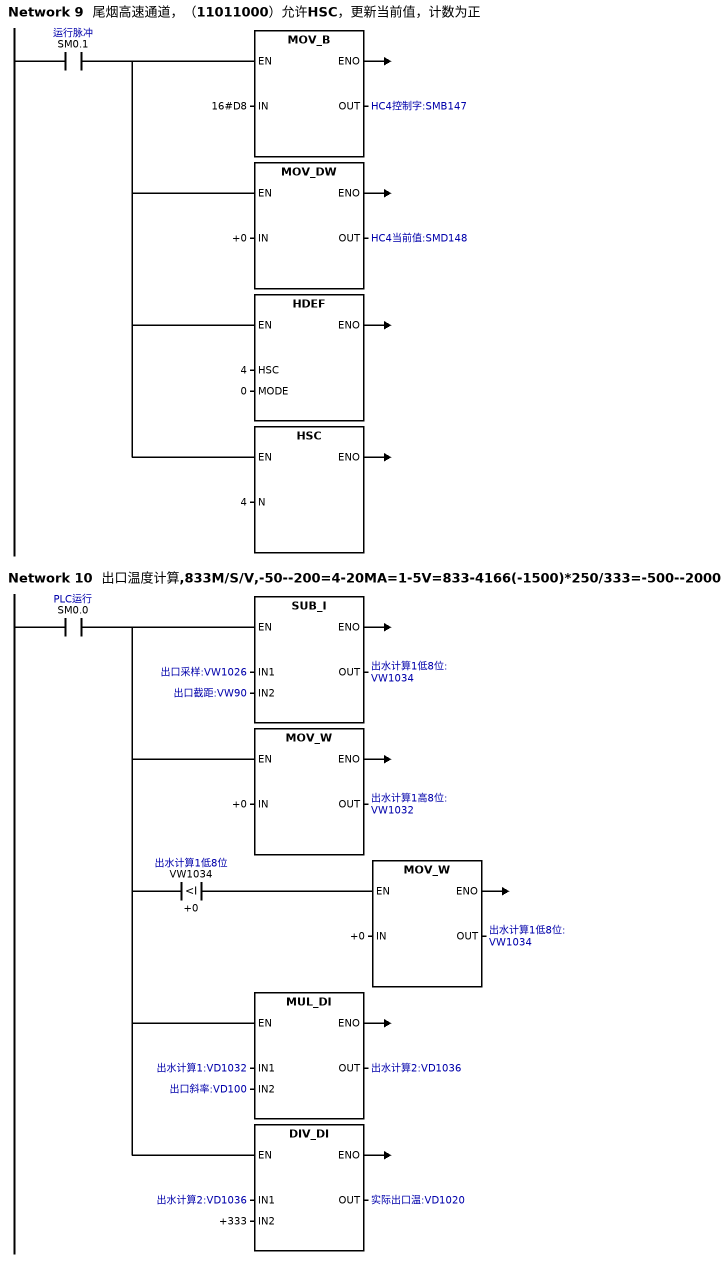
Network 9 // 尾烟高速通道，（11011000）允许HSC，更新当前值，计数为正
// 
// 
LD     运行脉冲:SM0.1
MOVB   16#D8, HC4控制字:SMB147
MOVD   +0, HC4当前值:SMD148
HDEF   4, 0
HSC    4
Network 10 // 出口温度计算,833M/S/V,-50--200=4-20MA=1-5V=833-4166(-1500)*250/333=-500--2000
// 
// 
LD     PLC运行:SM0.0
LPS
MOVW   出口采样:VW1026, 出水计算1低8位:VW1034
-I     出口截距:VW90, 出水计算1低8位:VW1034
MOVW   +0, 出水计算1高8位:VW1032
AW<    出水计算1低8位:VW1034, +0
MOVW   +0, 出水计算1低8位:VW1034
LRD
MOVD   出水计算1:VD1032, 出水计算2:VD1036
*D     出口斜率:VD100, 出水计算2:VD1036
LPP
MOVD   出水计算2:VD1036, 实际出口温:VD1020
/D     +333, 实际出口温:VD1020
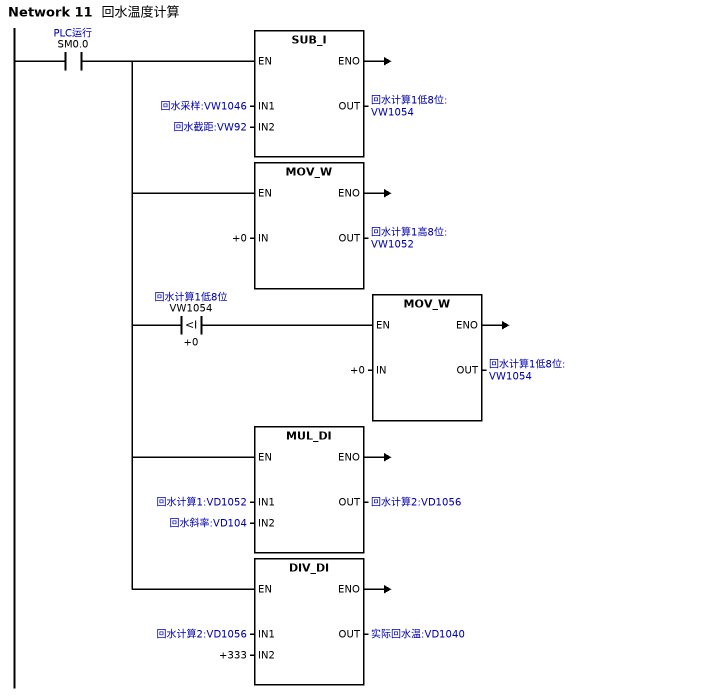
Network 11 // 回水温度计算
// 
// 
LD     PLC运行:SM0.0
LPS
MOVW   回水采样:VW1046, 回水计算1低8位:VW1054
-I     回水截距:VW92, 回水计算1低8位:VW1054
MOVW   +0, 回水计算1高8位:VW1052
AW<    回水计算1低8位:VW1054, +0
MOVW   +0, 回水计算1低8位:VW1054
LRD
MOVD   回水计算1:VD1052, 回水计算2:VD1056
*D     回水斜率:VD104, 回水计算2:VD1056
LPP
MOVD   回水计算2:VD1056, 实际回水温:VD1040
/D     +333, 实际回水温:VD1040
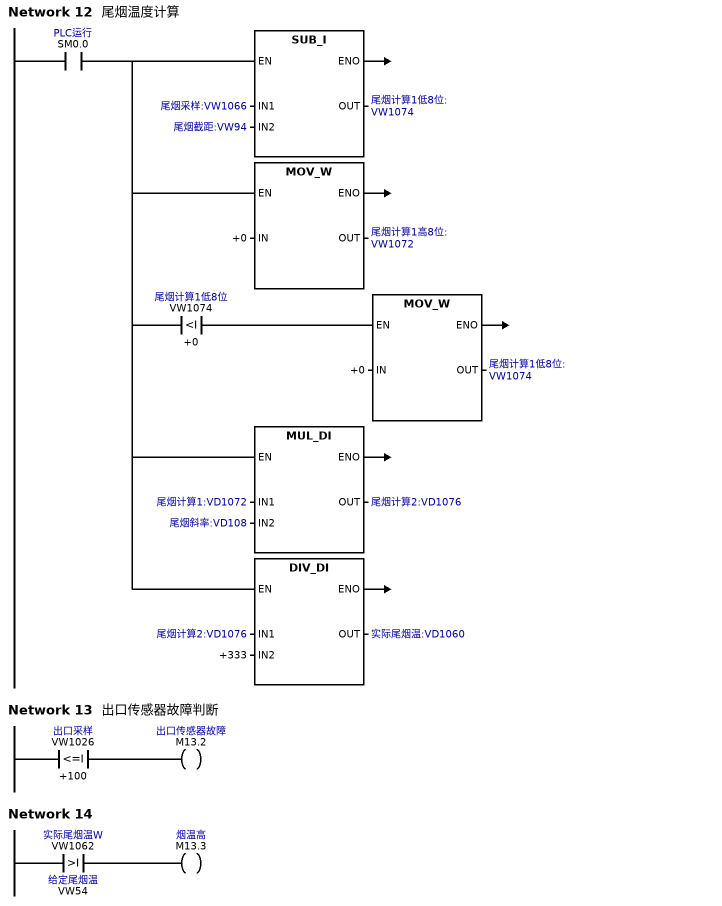
Network 12 // 尾烟温度计算
// 
// 
LD     PLC运行:SM0.0
LPS
MOVW   尾烟采样:VW1066, 尾烟计算1低8位:VW1074
-I     尾烟截距:VW94, 尾烟计算1低8位:VW1074
MOVW   +0, 尾烟计算1高8位:VW1072
AW<    尾烟计算1低8位:VW1074, +0
MOVW   +0, 尾烟计算1低8位:VW1074
LRD
MOVD   尾烟计算1:VD1072, 尾烟计算2:VD1076
*D     尾烟斜率:VD108, 尾烟计算2:VD1076
LPP
MOVD   尾烟计算2:VD1076, 实际尾烟温:VD1060
/D     +333, 实际尾烟温:VD1060
Network 13 // 出口传感器故障判断
// 
// 
LDW<=  出口采样:VW1026, +100
=      出口传感器故障:M13.2
Network 14
LDW>   实际尾烟温W:VW1062, 给定尾烟温:VW54
=      烟温高:M13.3
END_SUBROUTINE_BLOCK

// SBR1: protected block, not included

// SBR2: protected block, not included

// SBR3: protected block, not included

SUBROUTINE_BLOCK 故障检测:SBR4
TITLE= 
// SUBROUTINE COMMENTS
// Press F1 for help and example program
//  
BEGIN
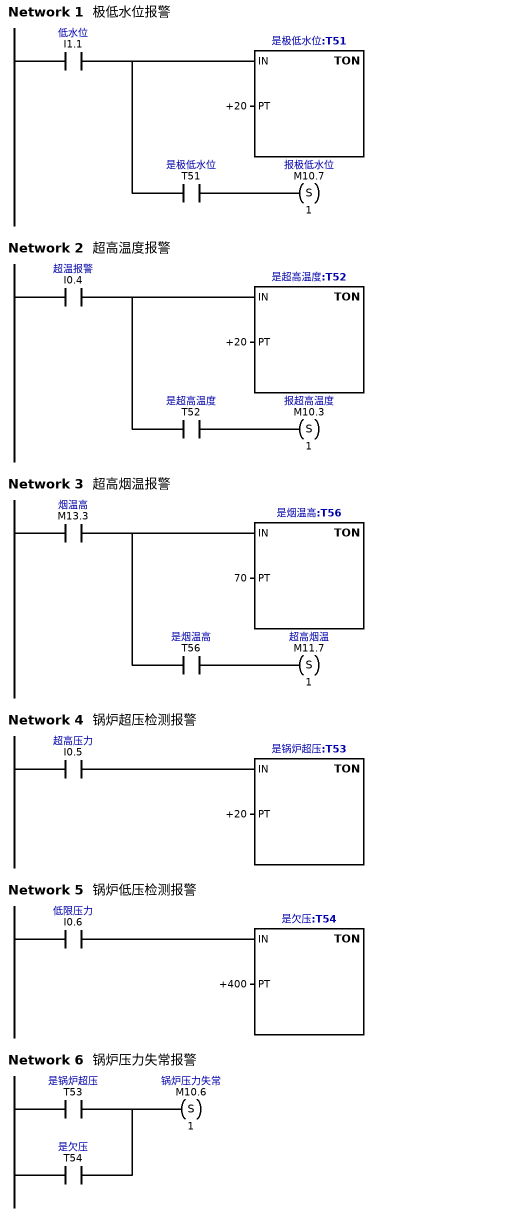
Network 1 // 极低水位报警
// 
// 
LD     低水位:I1.1
TON    是极低水位:T51, +20
A      是极低水位:T51
S      报极低水位:M10.7, 1
Network 2 // 超高温度报警
// 
// 
LD     超温报警:I0.4
TON    是超高温度:T52, +20
A      是超高温度:T52
S      报超高温度:M10.3, 1
Network 3 // 超高烟温报警
LD     烟温高:M13.3
TON    是烟温高:T56, 70
A      是烟温高:T56
S      超高烟温:M11.7, 1
Network 4 // 锅炉超压检测报警
// 
// 
LD     超高压力:I0.5
TON    是锅炉超压:T53, +20
Network 5 // 锅炉低压检测报警
// 
// 
LD     低限压力:I0.6
TON    是欠压:T54, +400
Network 6 // 锅炉压力失常报警
// 
// 
LD     是锅炉超压:T53
O      是欠压:T54
S      锅炉压力失常:M10.6, 1
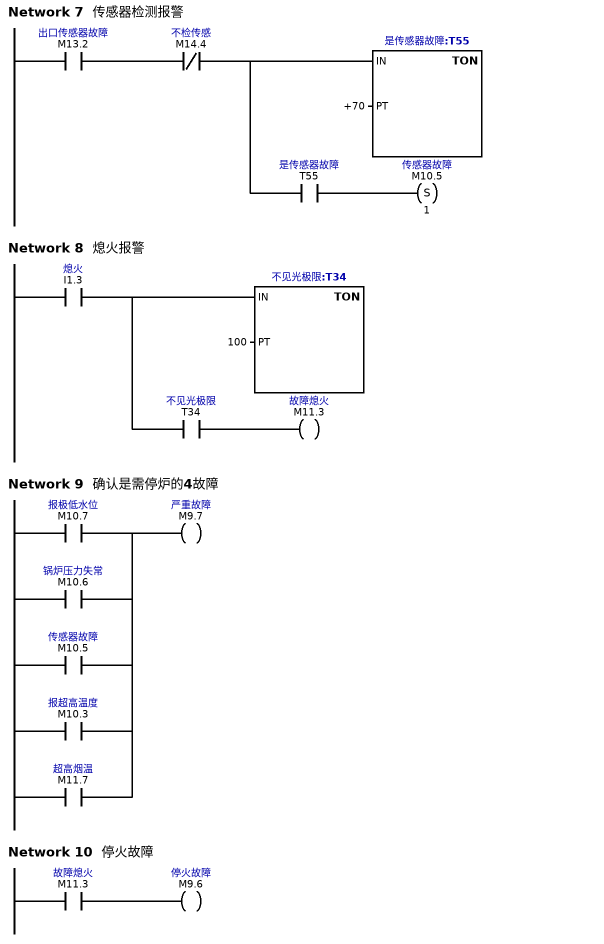
Network 7 // 传感器检测报警
// 
// 
LD     出口传感器故障:M13.2
AN     不检传感:M14.4
TON    是传感器故障:T55, +70
A      是传感器故障:T55
S      传感器故障:M10.5, 1
Network 8 // 熄火报警
// 
// 
LD     熄火:I1.3
TON    不见光极限:T34, 100
A      不见光极限:T34
=      故障熄火:M11.3
Network 9 // 确认是需停炉的4故障
// 
// 
LD     报极低水位:M10.7
O      锅炉压力失常:M10.6
O      传感器故障:M10.5
O      报超高温度:M10.3
O      超高烟温:M11.7
=      严重故障:M9.7
Network 10 // 停火故障
LD     故障熄火:M11.3
=      停火故障:M9.6
END_SUBROUTINE_BLOCK

SUBROUTINE_BLOCK 时间分段控制:SBR6
TITLE= 
// SUBROUTINE COMMENTS
// Press F1 for help and example program
BEGIN
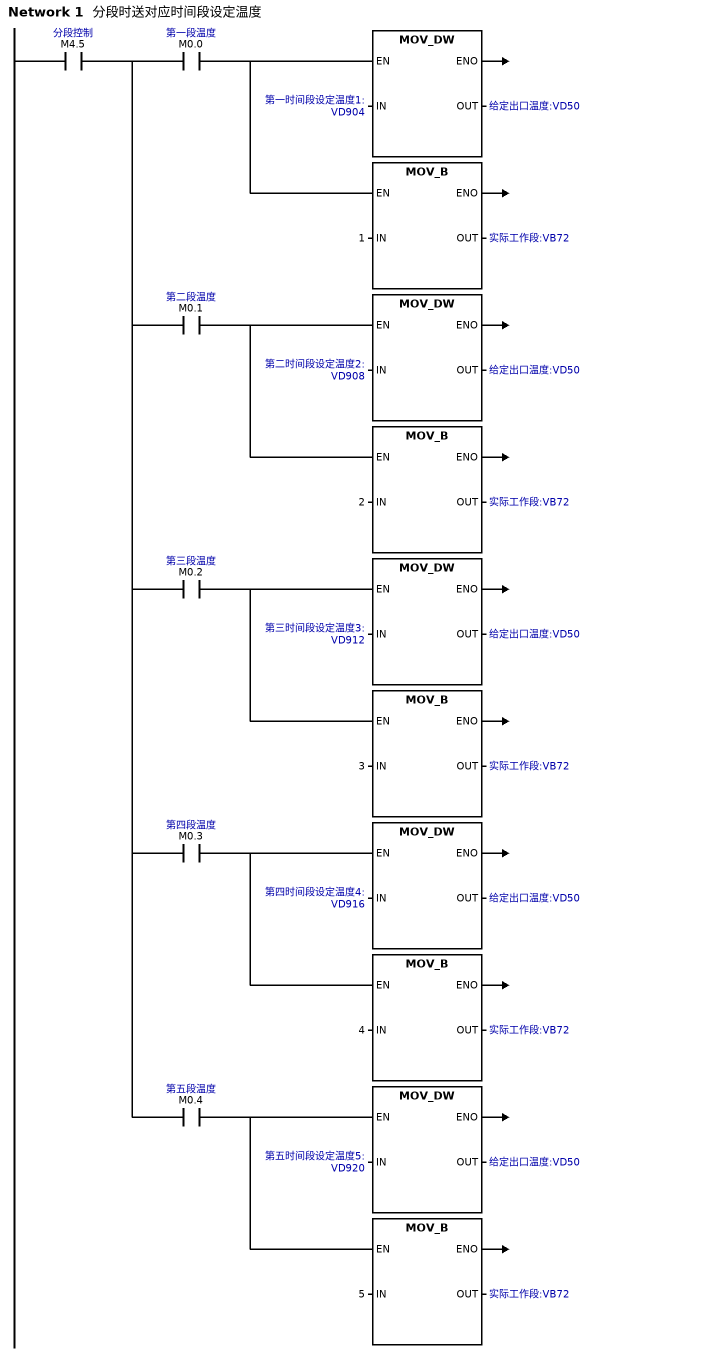
Network 1 // 分段时送对应时间段设定温度
LD     分段控制:M4.5
LPS
A      第一段温度:M0.0
MOVD   第一时间段设定温度1:VD904, 给定出口温度:VD50
MOVB   1, 实际工作段:VB72
LRD
A      第二段温度:M0.1
MOVD   第二时间段设定温度2:VD908, 给定出口温度:VD50
MOVB   2, 实际工作段:VB72
LRD
A      第三段温度:M0.2
MOVD   第三时间段设定温度3:VD912, 给定出口温度:VD50
MOVB   3, 实际工作段:VB72
LRD
A      第四段温度:M0.3
MOVD   第四时间段设定温度4:VD916, 给定出口温度:VD50
MOVB   4, 实际工作段:VB72
LPP
A      第五段温度:M0.4
MOVD   第五时间段设定温度5:VD920, 给定出口温度:VD50
MOVB   5, 实际工作段:VB72
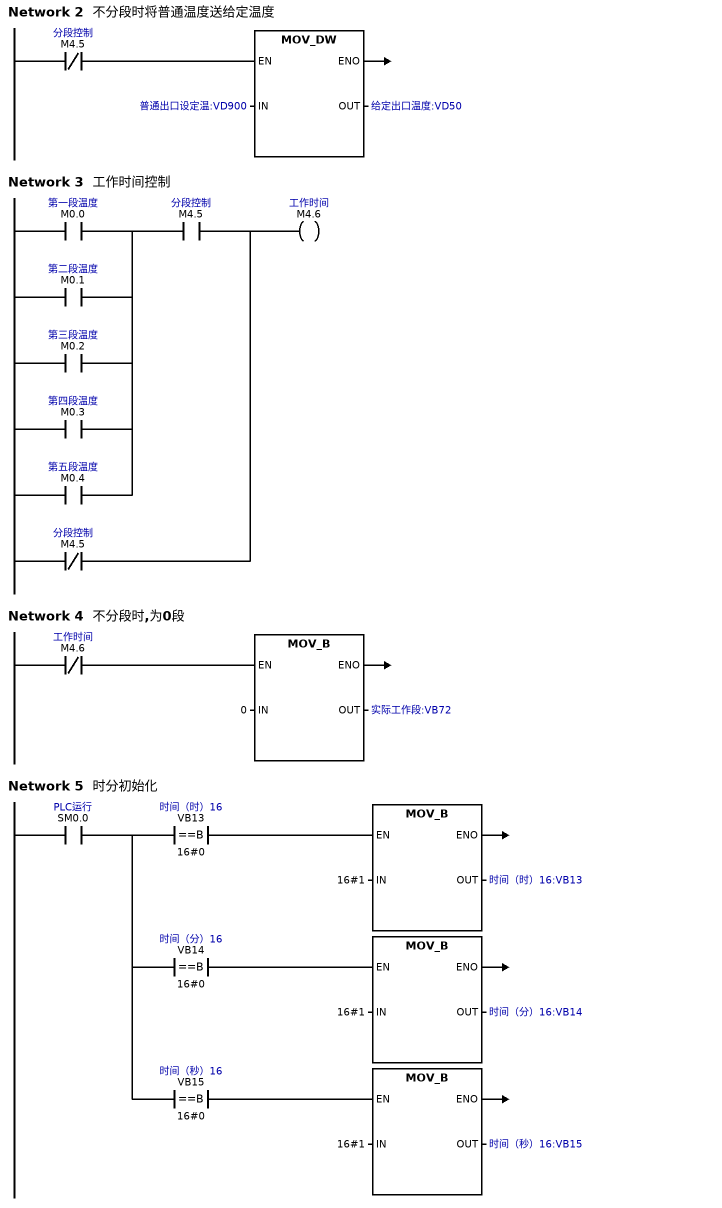
Network 2 // 不分段时将普通温度送给定温度
// 
// 
LDN    分段控制:M4.5
MOVD   普通出口设定温:VD900, 给定出口温度:VD50
Network 3 // 工作时间控制
// 
// 
LD     第一段温度:M0.0
O      第二段温度:M0.1
O      第三段温度:M0.2
O      第四段温度:M0.3
O      第五段温度:M0.4
A      分段控制:M4.5
ON     分段控制:M4.5
=      工作时间:M4.6
Network 4 // 不分段时,为0段
LDN    工作时间:M4.6
MOVB   0, 实际工作段:VB72
Network 5 // 时分初始化
LD     PLC运行:SM0.0
LPS
AB=    时间（时）16:VB13, 16#0
MOVB   16#1, 时间（时）16:VB13
LRD
AB=    时间（分）16:VB14, 16#0
MOVB   16#1, 时间（分）16:VB14
LPP
AB=    时间（秒）16:VB15, 16#0
MOVB   16#1, 时间（秒）16:VB15
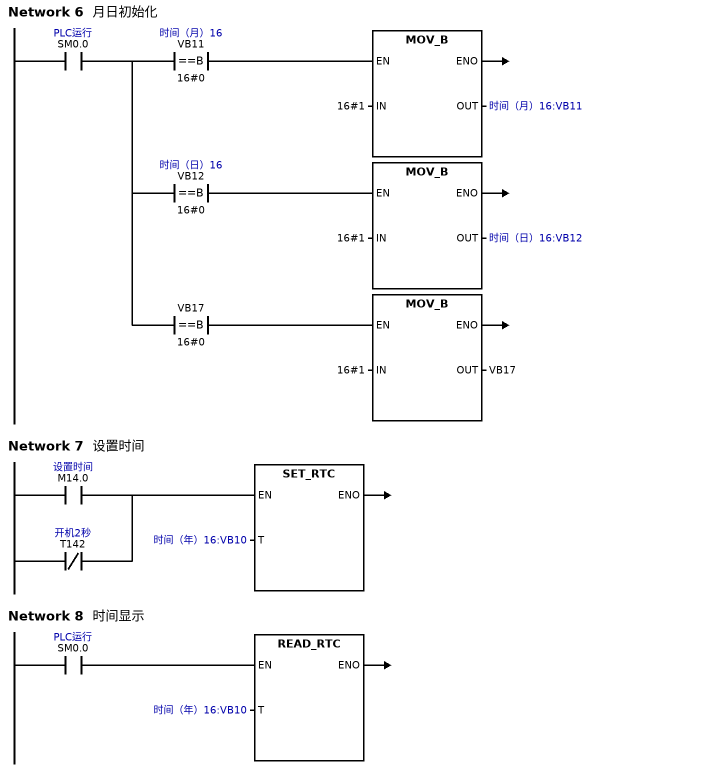
Network 6 // 月日初始化
LD     PLC运行:SM0.0
LPS
AB=    时间（月）16:VB11, 16#0
MOVB   16#1, 时间（月）16:VB11
LRD
AB=    时间（日）16:VB12, 16#0
MOVB   16#1, 时间（日）16:VB12
LPP
AB=    VB17, 16#0
MOVB   16#1, VB17
Network 7 // 设置时间
// 
// 
LD     设置时间:M14.0
ON     开机2秒:T142
TODW   时间（年）16:VB10
Network 8 // 时间显示
// 
// 
LD     PLC运行:SM0.0
TODR   时间（年）16:VB10
END_SUBROUTINE_BLOCK

SUBROUTINE_BLOCK 状态列表:SBR7
TITLE= 
// SUBROUTINE COMMENTS
// Press F1 for help and example program
//  
BEGIN
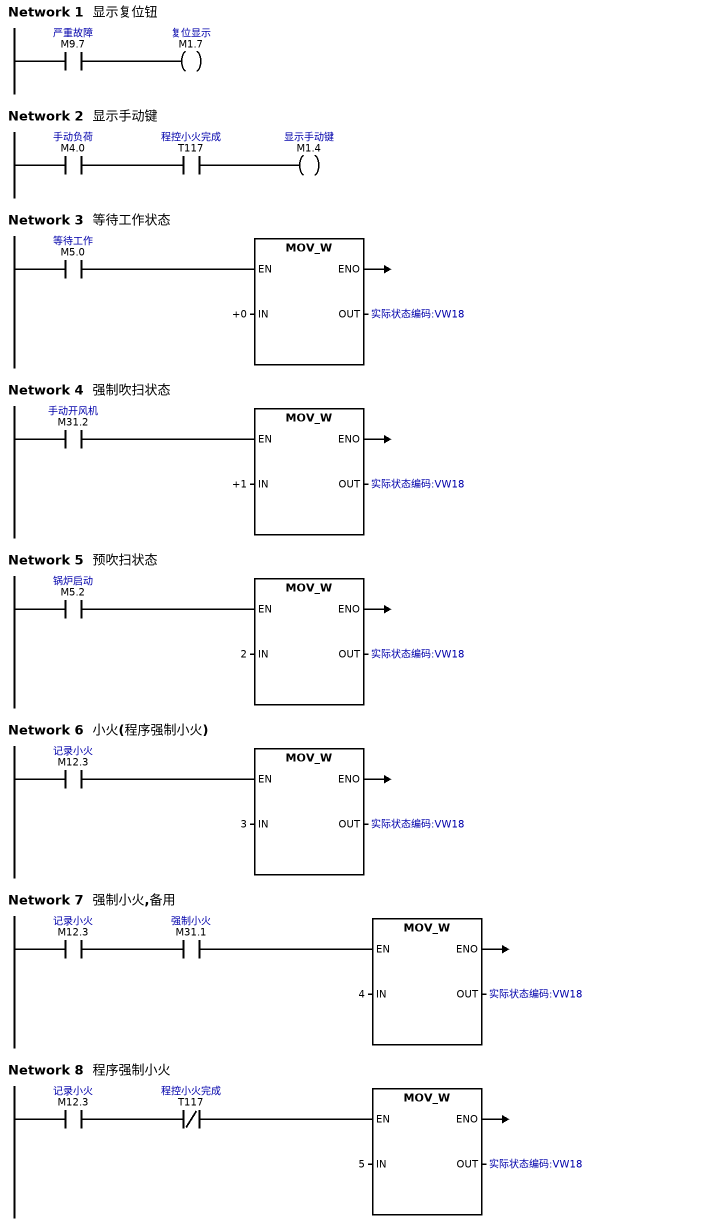
Network 1 // 显示复位钮
// 
//  
LD     严重故障:M9.7
=      复位显示:M1.7
Network 2 // 显示手动键
LD     手动负荷:M4.0
A      程控小火完成:T117
=      显示手动键:M1.4
Network 3 // 等待工作状态
// 
// 
LD     等待工作:M5.0
MOVW   +0, 实际状态编码:VW18
Network 4 // 强制吹扫状态
// 
// 
LD     手动开风机:M31.2
MOVW   +1, 实际状态编码:VW18
Network 5 // 预吹扫状态
// 
// 
LD     锅炉启动:M5.2
MOVW   2, 实际状态编码:VW18
Network 6 // 小火(程序强制小火)
LD     记录小火:M12.3
MOVW   3, 实际状态编码:VW18
Network 7 // 强制小火,备用
LD     记录小火:M12.3
A      强制小火:M31.1
MOVW   4, 实际状态编码:VW18
Network 8 // 程序强制小火
// 
// 
LD     记录小火:M12.3
AN     程控小火完成:T117
MOVW   5, 实际状态编码:VW18
